TYPE T_HMI_PACK_Barcode : STRING(cMAX_HMI_PACKCODE_LENGHT);
END_TYPE

(* stored: Version 1.1.0.1
   DUT T_HMI_PACK_Barcode: Id {87d9f579-d014-445b-83cf-1fb3312f62c9} *)
